// TwinCAT 3 PLC project LM_K2P3_PLC
// ProgramVersion: 3.1.4023.0
// libraries:
//   Tc2_Standard, * (Beckhoff Automation GmbH)
//   Tc2_System, * (Beckhoff Automation GmbH)
//   Tc3_Module, * (Beckhoff Automation GmbH)
// project tree:
//   / PlcTask.TcTTO
//   POUs/Alarms/ Alarm_Display_ST.TcPOU, Alarm_Flag.TcPOU, EtherCAT_Diagnostic.TcPOU
//   POUs/Main POUs/ Main.TcPOU, POU_Manual_Auto.TcPOU, POU_GatewaySignals.TcPOU, POU_Output.TcPOU
//   POUs/StateMachine_AutoManual/ AutoStates_POU.TcPOU
//   POUs/StateMachine_LaserMarking/ LaserMarking_Variable_Selection.TcPOU, LM_State_MC_TCP.TcPOU
//   POUs/StateMachine_MC_Axis/ MC_State_MC.TcPOU

CONFIGURATION LM_K2P3_PLC
    RESOURCE PLC ON TwinCAT3
        TASK PlcTask(INTERVAL := T#10ms, PRIORITY := 20);
        PROGRAM MAIN WITH PlcTask : MAIN;
    END_RESOURCE
END_CONFIGURATION

// ---- POUs/Main POUs/Main.TcPOU
PROGRAM Main
VAR
END_VAR

END_PROGRAM

// ---- POUs/Alarms/Alarm_Display_ST.TcPOU
PROGRAM Alarm_Display_ST
VAR
END_VAR

END_PROGRAM

// ---- POUs/Alarms/Alarm_Flag.TcPOU
PROGRAM Alarm_Flag
VAR
END_VAR

// NETWORK 1

END_PROGRAM

// ---- POUs/Alarms/EtherCAT_Diagnostic.TcPOU
PROGRAM EtherCAT_Diagnostic
VAR
END_VAR

END_PROGRAM

// ---- POUs/Main POUs/POU_Manual_Auto.TcPOU
PROGRAM POU_Manual_Auto
VAR
END_VAR

// NETWORK 1

END_PROGRAM

// ---- POUs/Main POUs/POU_GatewaySignals.TcPOU
PROGRAM POU_GatewaySignals
VAR
END_VAR

// NETWORK 1

END_PROGRAM

// ---- POUs/Main POUs/POU_Output.TcPOU
PROGRAM POU_Output
VAR
END_VAR
//tower Lamp POU

// NETWORK 1

END_PROGRAM

// ---- POUs/StateMachine_AutoManual/AutoStates_POU.TcPOU
PROGRAM AutoStates_POU
VAR
END_VAR

END_PROGRAM

// ---- POUs/StateMachine_LaserMarking/LaserMarking_Variable_Selection.TcPOU
PROGRAM LaserMarking_Variable_Selection
VAR
END_VAR

END_PROGRAM

// ---- POUs/StateMachine_LaserMarking/LM_State_MC_TCP.TcPOU
PROGRAM LM_State_MC_TCP
VAR
END_VAR

// NETWORK 1

END_PROGRAM

// ---- POUs/StateMachine_MC_Axis/MC_State_MC.TcPOU
PROGRAM MC_State_MC
VAR
END_VAR

// NETWORK 1

END_PROGRAM
